FUNCTION "m7a_1_OF_4_BITS" : VOID
TITLE =1 AUS 4 Bits: lässt nur 1 von 4 Bits mit High-Signal zu
//1 AUS 4 Bits: lässt nur 1 von 4 Bits mit High-Signal zu. Das letzte Signal mit
//positiver Flanke bleibt jeweils erhalten, die anderen beiden werden
//zurückgesetzt.
//
//VERWENDUNG:
//Richtungs- bzw. Positions- Steuersignale aus Schrittketten. Somit muss nur der
//jeweils aktuelle Richtungsmerker gesetzt werden, ohne den alten Richtungsmerker
//zu löschen. Dies hilft Flüchtigkeitsfehler bei Programmierung zu vermeiden.
//
//z.B. hat man eine Bewegung die mit 2 ungleich langen Zylindern auf 4 Positionen
//gesteuert wird:
//Positionen LINKS, MITTE_LINKS, MITTE_RECHTS, RECHTS. Ohne Verwendung dieses FCs
//muß man bei einem
//Positionswchsel immer alle 3 Richtungsmerker bearbeiten
//  S LINKS
//  R MITTE_LINKS
//  R MITTE_RECHTS
//  R RECHTS
//Mit Verwendung dieses FCs entfällt das Rücksetzen, somit ergibt sich als
//Steuerprogramm für LINKS nur noch
//  S LINKS
//
//AUTOR: Stefan Maag, Dipl.-Ing. (FH) Elektrotechnik
//DATUM: 9/2004
//INTERNET: www.maagic7.de
//
//AENDERUNGSVERMERKE:
//--------------------------------------------------------------------------------
//DATUM        NAME        AENDERUNG
//--------------------------------------------------------------------------------
//21.04.2009   S.Maag      FC-ENO-Ausgang := ein Eingangsbit ist aktiv
//
//05.01.2015   S.Maag      Flankenmerker zusammen mit Bits löschen sonst können 2
//                         Bits aktiv werden, wenn ein gelöschtes Bit im gleichen
//                         CPU Zyklus sofort wieder gesetzt wird.
//                         (kommt normal nicht vor und wie man sieht ist es
//                         erst nach 10Jahren aufgefallen!)
//--------------------------------------------------------------------------------
//
//HINWEISE:
AUTHOR : 'S.Maag'
FAMILY : Maagic7
VERSION : 0.1


VAR_IN_OUT
  Bit1 : BOOL ;	//Merker 1
  Bit2 : BOOL ;	//Merker 2
  Bit3 : BOOL ;	//Merker 3
  Bit4 : BOOL ;	//Merker 4
  tmpByte : BYTE ;	//Hilfsbyte für Zustandsspeicherung
END_VAR
VAR_TEMP
  tmpBit1 : BOOL ;
  tmpBit2 : BOOL ;
  tmpBit3 : BOOL ;
  tmpBit4 : BOOL ;
  tmpBit5 : BOOL ;
  tmpBit6 : BOOL ;
  tmpBit7 : BOOL ;
  tmpBit8 : BOOL ;
END_VAR
BEGIN
NETWORK
TITLE =Hilfsbyte in lokalen Speicherbereich zur Bitadressierung

      L     #tmpByte;
      T     LB     0;
NETWORK
TITLE =Flanken der Bits prüfen und andere Bits löschen

      U     #Bit1; // Bit 1 auf positive Flanke prüfen
      FP    #tmpBit1;
      SPB   C234; // wenn ja, Bit 2/3/4 löschen

      U     #Bit2; // Bit 2 auf positive Flanke prüfen
      FP    #tmpBit2;
      SPB   C134; // wenn ja, Bit 1/3/4 löschen

      U     #Bit3;
      FP    #tmpBit3;
      SPB   C124;

      U     #Bit4;
      FP    #tmpBit4;
      SPB   C123;
      SPA   END;

C234: R     #Bit2; // CLR Bit 2/3/4
      R     #Bit3;
      R     #Bit4;
      R     #tmpBit2; // CLR Flankenmerker
      R     #tmpBit3; // CLR Flankenmerker
      R     #tmpBit4; // CLR Flankenmerker
      SPA   END;
C134: R     #Bit1; // CLR Bit 1/3/4
      R     #Bit3;
      R     #Bit4;
      R     #tmpBit1; // CLR Flankenmerker
      R     #tmpBit3; // CLR Flankenmerker
      R     #tmpBit4; // CLR Flankenmerker
      SPA   END;
C124: R     #Bit1; // CLR Bit 1/2/4
      R     #Bit2;
      R     #Bit4;
      R     #tmpBit1; // CLR Flankenmerker
      R     #tmpBit2; // CLR Flankenmerker
      R     #tmpBit4; // CLR Flankenmerker
      SPA   END;
C123: R     #Bit1; // CLR Bit 1/2/3
      R     #Bit2;
      R     #Bit3;
      R     #tmpBit1; // CLR Flankenmerker
      R     #tmpBit2; // CLR Flankenmerker
      R     #tmpBit3; // CLR Flankenmerker

NETWORK
TITLE =aktuelles Hilfsbyte wieder zurückschreiben

END:  L     LB     0;
      T     #tmpByte;

      O     #Bit1;
      O     #Bit2;
      O     #Bit3;
      O     #Bit4;
      SAVE  ;
      CLR   ;

END_FUNCTION

FUNCTION "m7a_CreateS5TimeFromINT" : VOID
TITLE =Minuten, Sekunden (im INT-Format) in das S5Time-Format wandeln
//Umwandlung von Minuten und/oder Sekunden in das S5Time-Format mit der
//gümstigsten Zeitbasis.
//Maximal sind mit dem S5Time-Format 9990sec möglich, das entspricht 2h46min30sec
//oder 166min 30sec
//
//AUTOR: Stefan Maag, Dipl.-Ing. (FH) Elektrotechnik
//DATUM: 9/2004
//INTERNET: www.maagic7.de
//
//AENDERUNGSVERMERKE:
//--------------------------------------------------------------------------------
//DATUM        NAME        AENDERUNG
//--------------------------------------------------------------------------------
//24.01.2005   S.Maag    Fehler BCD Wandlung bei Zeitbasis 10sec behoben
//--------------------------------------------------------------------------------
//
//HINWEISE:
AUTHOR : 'S.Maag'
FAMILY : Maagic7
VERSION : 0.1


VAR_INPUT
  MIN : INT ;	//Anzahl Minuten (max = 166min, da S5MaxTime=9990sec)
  SEC : INT ;	//Anzahl Sekunden
END_VAR
VAR_OUTPUT
  S5_TIME : S5TIME ;
END_VAR
BEGIN
NETWORK
TITLE =Umwandlung in die günstigste Zeitbasis
//S5Time-Format Bits:
//
//15 | 14 | 13 | 12 | 11 | 10 | 9 | 8 | 7 | 6 | 5 | 4 | 3 | 2 | 1 | 0
//  x   x | Zeitbas.|             Zeitwert im BCD Format
//
//Zeitbasis : Bits fuer Zeitbasis
//     10ms : 00
//    100ms : 01
//      1s  : 10
//     10s  : 11
      L     #MIN; // Minuten
      L     60; // Sekunden/Minute
      *I    ; // Sekunden von Minuten
      L     #SEC; // Sekunden
      +I    ; // Sekunden gesamt
      L     9; // bis 9 Sekunden
      TAK   ; // Sekunden in Akku 1, Vergleichswert in Akku 2
      >=I   ;
      SPB   hdst; // Zeitbasis 10ms = 1/100sec

      L     99; // bis 99 Sekunden
      TAK   ;
      >=I   ;
      SPB   zntl; // Zeitbasis 100ms = 1/10sec

      L     990; // bis 990 Sekunden
      TAK   ;
      >=I   ;
      SPB   sec; // Zeitbasis 1 Sekunde

      L     9990;
      TAK   ;
      >=I   ; // falls nicht mehr als 9990 Sekunden, dann
      SPB   zehn; // Zeitbasis Zehn Sekunden
      TAK   ; // sonst Begrenzung: 9990 wieder in Akku 1

zehn: L     10; // zuerst durch 10 teilen, da  Werte > 999 nicht mit
      /I    ; // dem ITB Befehl in BCD gewandelt werden können. Ein SRW 4 der
      ITB   ; // BCD Zahl geht hier nicht, da die Sekunden > 999 sein können.
      L     W#16#3000; // Zeitbasis Zehn Sekunden
      OW    ; // Bits für Zeitbasis einblenden
      SPA   SAVE;

sec:  ITB   ; // Anzahl der Sekunden ins BCD Format
      L     W#16#2000; // Zeitbasis Sekunden
      OW    ; // Bits für Zeitbasis einblenden
      SPA   SAVE;

zntl: ITB   ; // Anzahl der Sekunden (max, 999) ins BCD Format
      SLW   4; // 4 Bits nach links := 1 Stelle im 10er BCD Format := *10
      L     W#16#1000; // Zeitbasis 10ms
      OW    ; // Bits für Zeitbasis einblenden
      SPA   SAVE;

hdst: ITB   ; // Anzahl der Sekunden ins BCD Format
      SLW   8; // 8 Bits nach links := 2 Stellen im 10er BCD Format := *100
      L     W#16#0; // Zeitbasis 100ms
      OW    ; // Bits für Zeitbasis einblenden
SAVE: T     #S5_TIME; // Zeit im S5Time-Format
NETWORK
TITLE =FC-ENO

      SET   ;
      SAVE  ;
      CLR   ;

END_FUNCTION

FUNCTION "m7a_CreateIECTimeFromINT" : VOID
TITLE =Time hh:mm:ss [INT] to IEC TIME
//AUTOR: Stefan Maag, Dipl.-Ing. (FH) Elektrotechnik
//DATUM: 9/2004
//INTERNET: www.maagic7.de
//
//AENDERUNGSVERMERKE:
//--------------------------------------------------------------------------------
//DATUM        NAME        AENDERUNG
//--------------------------------------------------------------------------------
//20.03.2018   S.Maag      changed from mm:ss to hh:mm:ss
//--------------------------------------------------------------------------------
//
//HINWEISE:
AUTHOR : 'S.Maag'
FAMILY : Maagic7
VERSION : 0.1


VAR_INPUT
  hh : INT ;	//Hours
  mm : INT ;	//Minutes
  ss : INT ;	//Seconds
END_VAR
VAR_OUTPUT
  IEC_TIME : TIME ;
END_VAR
VAR_TEMP
  dMilliSeconds : DINT ;	//Sekunden als Millisekunden
END_VAR
BEGIN
NETWORK
TITLE =ss to milli seconds

      L     #ss; // seconds
      ITD   ; // to DINT
      L     L#1000; // 1sec = 1000ms
      *D    ;
      T     #dMilliSeconds; // save

NETWORK
TITLE =Minutes to milli seconds

      L     #mm; // Minutes
      ITD   ; // to DINT
      L     L#60000; // 1 min = 60000ms
      *D    ;
      L     #dMilliSeconds;
      +D    ;
      T     #dMilliSeconds;

NETWORK
TITLE =hours to milli seconds

      L     #hh; // hours
      ITD   ; // to DINT
      L     L#3600000; // 1h = 3600.000ms
      *D    ;
      L     #dMilliSeconds;
      +D    ;
      T     #IEC_TIME;

NETWORK
TITLE =FC-ENO-Ausgang

      SET   ;
      SAVE  ;
      CLR   ;

END_FUNCTION

FUNCTION "m7a_INV_IEC_TIME" : VOID
TITLE =IEC Zeit invertieren, Rückwärtszählung
//IEC Zeit invertieren. Wird benötigt z.B. benötigt, wenn Ausschaltverzögerungen
//über SFB5 programmiert werden und die Zeitanzeige dann rückwärts laufen soll.
//SFB5 stellt nur einen vorwärts laufenden Timerwert zur Verfügung
//
//AUTOR: Stefan Maag, Dipl.-Ing. (FH) Elektrotechnik
//DATUM: 1/2005
//INTERNET: www.maagic7.de
//
//AENDERUNGSVERMERKE:
//--------------------------------------------------------------------------------
//DATUM        NAME            AENDERUNG
//--------------------------------------------------------------------------------
//
//--------------------------------------------------------------------------------
//
//HINWEISE:
AUTHOR : 'S.Maag'
FAMILY : Maagic7
VERSION : 0.1


VAR_INPUT
  iecDauer : TIME ;	//Dauer
  iecTimer : TIME ;	//Zeitwert vom Timer
END_VAR
VAR_OUTPUT
  iecInvTime : TIME ;
END_VAR
BEGIN
NETWORK
TITLE =

      L     #iecDauer;
      L     #iecTimer;
      -D    ;
      L     L#0;
      <D    ;
      SPB   SAVE;
      TAK   ;
SAVE: T     #iecInvTime;
NETWORK
TITLE =FC-ENO

      SET   ;
      SAVE  ;
      CLR   ;

END_FUNCTION

FUNCTION "m7a_DINT_MM.SS_TO_IEC" : VOID
TITLE =Zeit DINT MM.SS in das IEC-Zeitformat wandeln
//AUTOR: Stefan Maag, Dipl.-Ing. (FH) Elektrotechnik
//DATUM: 1/2005
//INTERNET: www.maagic7.de
//
//AENDERUNGSVERMERKE:
//--------------------------------------------------------------------------------
//DATUM        NAME       AENDERUNG
//--------------------------------------------------------------------------------
//22.04.2014   S.Maag     Ausgang IEC-Zeit auf min. 1ms begrenzt, da 0ms = RESET
//--------------------------------------------------------------------------------
//
//HINWEISE:
AUTHOR : 'S.Maag'
FAMILY : Maagic7
VERSION : 0.1


VAR_OUTPUT
  IEC_TIME : TIME ;
END_VAR
VAR_IN_OUT
  MM_SS : DINT ;	//Minuten und Sekunden z.B.: 0530 = 5m30s
END_VAR
VAR_TEMP
  MM : DINT ;	//Minutenwert
  SS : DINT ;	//Sekundenwert
  SS_msec : DINT ;	//Sekunden als Millisekunden
END_VAR
BEGIN
NETWORK
TITLE =Minuten und Sekundenanteil aus MM.SS lösen

      L     #MM_SS; // Minuten.Sekunden
      L     L#100;
      MOD   ; // Modulo Division
      T     #SS; // =Divisionsrest = Sekunden

      L     #MM_SS;
      L     L#100;
      /D    ;
      T     #MM;

NETWORK
TITLE =Sekundenanteil in Millisekunden umrechnen

      L     #SS; // Sekunden
      L     1000;
      *D    ;
      T     #SS_msec; // Millisekunden

NETWORK
TITLE =Minutenanteil in Millisekunden umrechnen
//22.04.2014 IEC-Zeit auf min. 1ms begrenzt, da 0ms = RESET
      L     #MM; // Minuten
      L     L#60000; // Millisekunden pro Minute
      *D    ;
      L     #SS_msec; // Anteil der Sekunden
      +D    ; // + Anteil der Minuten
      U     >0;
      SPB   save;
      L     L#1;
save: T     #IEC_TIME; // ergibt gesamte Millisekunden

NETWORK
TITLE =Wenn Sekunden >59, dann 1 Minute dazu und Sekunden anpassen

      L     #SS; // Sekundenwert
      L     59; // prüfen, ob weniger als 60
      <=D   ; // Sekunden, dann o.k.
      SPB   NE4;

      L     #MM_SS; // Minuten.Sekunden laden
      +     L#40; // Wenn mehr als 60Sekunden, dann müssen die fehlenden
      T     #MM_SS; // 40 Sekunden für den Überlauf dazugezählt werden
NE4:  NOP   0;

NETWORK
TITLE =FC-ENO-Ausgang

      SET   ;
      SAVE  ;
      CLR   ;

END_FUNCTION

FUNCTION "m7a_IEC_TO_MM.SS_DINT" : VOID
TITLE =IEC Zeit in DINT MM.SS wandeln
//AUTOR: Stefan Maag, Dipl.-Ing. (FH) Elektrotechnik
//DATUM: 1/2005
//INTERNET: www.maagic7.de
//
//AENDERUNGSVERMERKE:
//--------------------------------------------------------------------------------
//DATUM        NAME            AENDERUNG
//--------------------------------------------------------------------------------
//
//--------------------------------------------------------------------------------
//
//HINWEISE:
AUTHOR : 'S.Maag'
FAMILY : Maagic7
VERSION : 0.1


VAR_INPUT
  IEC_TIME : TIME ;
END_VAR
VAR_OUTPUT
  MM_SS : DINT ;
END_VAR
VAR_TEMP
  MM : DINT ;	//Minutenwert
  SS : DINT ;	//Sekundenwert
END_VAR
BEGIN
NETWORK
TITLE =Minuten- und Sekundenanteil

      L     #IEC_TIME;
      L     L#60000; // Millisekunden pro Minute
      /D    ;
      T     #MM; // Minuten

      L     #IEC_TIME;
      L     L#60000; // Millisekunden pro Minute
      MOD   ; // Restwerdivision: Rest ms
      L     L#1000;
      /D    ; // Modulo Division
      T     #SS; // =Divisionsrest = Sekunden

      L     #MM; // Minuten*100
      L     L#100;
      *D    ;
      L     #SS;
      +D    ;
      T     #MM_SS; // Wert in MM.SS

NETWORK
TITLE =FC-ENO-Ausgang

      SET   ;
      SAVE  ;
      CLR   ;

END_FUNCTION

FUNCTION "m7a_DINT_MM.SS_TO_S5Time" : VOID
TITLE =Zeit DINT MM.SS in das S5-Zeitformat wandeln
//Zeiten werden als DINT-Wert mit 2 Nachkommastellen eingegeben, welche den
//Sekunden entsprechen. Die Minuten sind der Wert vor dem Komma. Werden Sekunden
//größer als 59 eingegebn, so werden diese automatisch auf Minuten umgerechnet
//und der eingegebene Wert MM.SS richtig angepasst.
//
//AUTOR: Stefan Maag, Dipl.-Ing. (FH) Elektrotechnik
//DATUM: 1/2005
//INTERNET: www.maagic7.de
//
//AENDERUNGSVERMERKE:
//--------------------------------------------------------------------------------
//DATUM        NAME            AENDERUNG
//--------------------------------------------------------------------------------
//
//--------------------------------------------------------------------------------
//
//HINWEISE:
AUTHOR : 'S.Maag'
FAMILY : Maagic7
VERSION : 0.1


VAR_OUTPUT
  S5_Time : S5TIME ;
END_VAR
VAR_IN_OUT
  MM_SS : DINT ;	//Minuten und Sekunden z.B.: 0530 = 5m30s
END_VAR
VAR_TEMP
  MM : INT ;	//Minutenwert
  SS : INT ;	//Sekundenwert
END_VAR
BEGIN
NETWORK
TITLE =Minuten und Sekundenanteil aus MM.SS lösen

      L     #MM_SS; // Minuten.Sekunden
      L     L#100;
      MOD   ; // Modulo Division
      T     #SS; // =Divisionsrest = Sekunden

      L     #MM_SS;
      L     L#100;
      /D    ;
      T     #MM;

NETWORK
TITLE =Wenn Sekunden >59, dann 1 Minute dazu und Sekunden anpassen

      L     #SS; // Sekundenwert
      L     59; // prüfen, ob weniger als 60
      <=D   ; // Sekunden, dann o.k.
      SPB   NE4;

      L     #MM_SS; // Minuten.Sekunden laden
      +     L#40; // Wenn mehr als 60Sekunden, dann müssen die fehlenden
      T     #MM_SS; // 40 Sekunden für den Überlauf dazugezählt werden
NE4:  NOP   0;

NETWORK
TITLE =Umwandlung in die günstigste Zeitbasis
//S5Time-Format Bits:
//
//15 | 14 | 13 | 12 | 11 | 10 | 9 | 8 | 7 | 6 | 5 | 4 | 3 | 2 | 1 | 0
//  x   x | Zeitbas.|             Zeitwert im BCD Format
//
//Zeitbasis : Bits fuer Zeitbasis
//     10ms : 00
//    100ms : 01
//      1s  : 10
//     10s  : 11
      L     #MM; // Minuten
      L     60; // Sekunden/Minute
      *D    ; // Sekunden von Minuten
      L     #SS; // Sekunden
      +D    ; // Sekunden gesamt
      L     9; // bis 9 Sekunden
      TAK   ; // Sekunden in Akku 1, Vergleichswert in Akku 2
      >=I   ;
      SPB   hdst; // Zeitbasis 10ms = 1/100sec

      L     99; // bis 99 Sekunden
      TAK   ;
      >=I   ;
      SPB   zntl; // Zeitbasis 100ms = 1/10sec

      L     990; // bis 990 Sekunden
      TAK   ;
      >=I   ;
      SPB   sec; // Zeitbasis 1 Sekunde

      L     9990;
      TAK   ;
      >=I   ; // falls nicht mehr als 9990 Sekunden, dann
      SPB   zehn; // Zeitbasis Zehn Sekunden
      TAK   ; // sonst Begrenzung: 9990 wieder in Akku 1

zehn: L     10; // zuerst durch 10 teilen, da  Werte > 999 nicht mit
      /I    ; // dem ITB Befehl in BCD gewandelt werden können. Ein SRW 4 der
      ITB   ; // BCD Zahl geht hier nicht, da die Sekunden > 999 sein können.
      L     W#16#3000; // Zeitbasis Zehn Sekunden
      OW    ; // Bits für Zeitbasis einblenden
      SPA   SAVE;

sec:  ITB   ; // Anzahl der Sekunden ins BCD Format
      L     W#16#2000; // Zeitbasis Sekunden
      OW    ; // Bits für Zeitbasis einblenden
      SPA   SAVE;

zntl: ITB   ; // Anzahl der Sekunden (max, 999) ins BCD Format
      SLW   4; // 4 Bits nach links := 1 Stelle im 10er BCD Format := *10
      L     W#16#1000; // Zeitbasis 10ms
      OW    ; // Bits für Zeitbasis einblenden
      SPA   SAVE;

hdst: ITB   ; // Anzahl der Sekunden ins BCD Format
      SLW   8; // 8 Bits nach links := 2 Stellen im 10er BCD Format := *100
      L     W#16#0; // Zeitbasis 100ms
      OW    ; // Bits für Zeitbasis einblenden
SAVE: T     #S5_Time; // Zeit im S5Time-Format
NETWORK
TITLE =FC-ENO-Ausgang

      SET   ;
      SAVE  ;
      CLR   ;

END_FUNCTION

FUNCTION "m7a_MMSS_BCD_TO_IEC" : VOID
TITLE =Zeit hexadezimal MM.SS in das IEC-Zeitformat wandeln
//AUTOR: Stefan Maag, Dipl.-Ing. (FH) Elektrotechnik
//DATUM: 10/2004
//INTERNET: www.maagic7.de
//
//AENDERUNGSVERMERKE:
//--------------------------------------------------------------------------------
//DATUM        NAME        AENDERUNG
//--------------------------------------------------------------------------------
//
//--------------------------------------------------------------------------------
//
//HINWEISE:
AUTHOR : 'S.Maag'
FAMILY : Maagic7
VERSION : 0.1


VAR_INPUT
  MIN_BCD : BYTE ;	//Minuten als BCD-Wert
  SEC_BCD : BYTE ;	//Sekunden als BCD-Wert
END_VAR
VAR_OUTPUT
  IEC_TIME : TIME ;
END_VAR
VAR_TEMP
  SS_msec : DINT ;	//Sekunden als Millisekunden
END_VAR
BEGIN
NETWORK
TITLE =Sekundenanteil in Millisekunden umrechen

      L     #SEC_BCD; // Sekunden im HEX-Format
      SLD   12; // * 1000 = Millisekunden
      BTD   ; // BCD->DINT
      T     #SS_msec; // zwischenspeichern

NETWORK
TITLE =Minutenanteil in Millisekunden umrechnen

      L     #MIN_BCD; // Minuten im HEX-Format
      SLD   12; // *1000
      BTD   ; // BCD->DINT
      L     L#60; // Sekunden pro Minute
      *D    ; // *1000 *60 := Millisekunden
      L     #SS_msec; // Anteil der Sekunden
      +D    ; // + Anteil der Minuten
      T     #IEC_TIME; // ergibt gesamte Millisekunden

NETWORK
TITLE =FC-ENO-Ausgang

      SET   ;
      SAVE  ;
      CLR   ;

END_FUNCTION

FUNCTION "m7a_ZeitDauer" : VOID
TITLE =Zeitdauer Abgelaufen?
//Überprüft, ob seit der übergebenen Startzeit die gewünschte Dauer abgelaufen
//ist. Die Zeiten werden im IEC-TIME-FORMAT übergeben
//
//BENÖTIGTE SFCs: SFC1 - READ_CLK
//
//AUTOR: Stefan Maag, Dipl.-Ing. (FH) Elektrotechnik
//DATUM: 9/2004
//INTERNET: www.maagic7.de
//
//AENDERUNGSVERMERKE:
//--------------------------------------------------------------------------------
//DATUM        NAME        AENDERUNG
//--------------------------------------------------------------------------------
//03/12/2013   S.Maag      SFC64 TimeTick Zeitdifferenz korrigiert
//                         da 31Bit, Fehler bei Überlauf. Jetzt UC FC256
//--------------------------------------------------------------------------------
//
//HINWEISE:
AUTHOR : 'S.Maag'
FAMILY : Maagic7
VERSION : 0.1


VAR_INPUT
  START_ZEIT : TIME ;
  DAUER : TIME ;
END_VAR
VAR_OUTPUT
  OUT_TIMER : BOOL ;	//TimerAusgang: Zeit abgelaufen
  TIME_LEFT : TIME ;	//Restlaufzeit
END_VAR
VAR_TEMP
  aktSysTime : TIME ;	//aktuelle Systemzeit
END_VAR
BEGIN
NETWORK
TITLE =aktuelle SystemZeit auslesen

      CALL "TIME_TCK" (
           RET_VAL                  := #aktSysTime);
      NOP   0;

NETWORK
TITLE =prüfen ob Zeit abgelaufen ist

      L     #START_ZEIT;
      L     #aktSysTime;
      UC    "m7b_ABS_DIFF_S7SysTime"; // Absolute Differenz S7SytemTimer 31Bit
      L     #DAUER;
      >D    ;
      =     #OUT_TIMER;
      SAVE  ;
      TAK   ;
      -D    ;
      T     #TIME_LEFT;

END_FUNCTION

FUNCTION "m7a_CreateANY" : VOID
TITLE =CreateANY: erzeugt ANY aus Einzelbestandteilen
//Codierung Datentyp:
//00h : NIL  : Nullpointer
//01h : BOOL : Bits
//02h : BYTE
//03h : CHAR
//04h : WORD
//05h : INT
//06h : DWORD
//07h : DINT
//08h : REAL
//09h : DATE
//0Ah : Time_OF_DAY (TOD)
//0Bh : TIME
//0Ch : S5Time
//0Dh : nicht definiert
//0Eh : DATE_AND_TIME (DT)
//13h : STRING
//
//Codierung Speicherbereich:
//80h : P : Peripherie
//81h : E : Eingänge
//82h : A : Ausgänge
//83h : M : Merker
//84h : DB: Datenbaustein
//85h : DI: Instanzdatenbaustein
//86h : L : Lokaldaten (L-Stack)
//87h : V : voriger Lokaldatenstack
//
//AUTOR: Stefan Maag, Dipl.-Ing. (FH) Elektrotechnik
//DATUM: 10/2007
//INTERNET: www.maagic7.de
//
//AENDERUNGSVERMERKE:
//--------------------------------------------------------------------------------
//DATUM        NAME       AENDERUNG
//--------------------------------------------------------------------------------
//04.11.2011   S.Maag     Fehler Speicherbereichsverarbeitung mit UD statt OD
//                        behoben
//--------------------------------------------------------------------------------
//
//HINWEISE:
AUTHOR : 'S.Maag'
FAMILY : Maagic7
VERSION : 0.1


VAR_INPUT
  B1_DataType : BYTE ;	//1=Bool 2=Byte 3=Char 4=Word 5=INT 6=DW 7=DINT 8=Real 9=Date ...
  B23_Wiederholung : INT ;	//Wiederholungsfaktor
  B45_DB : INT ;	//DB-Nummer oder 0
  B6_Speicher : BYTE ;	//Hex 80=P 81=E 82=A 83=M 84=DB 85=DI 86=L 87=V
  ByteAdr : INT ;	//ByteAdresse
  BitAdr : INT ;	//Bitadresse 0..7
END_VAR
VAR_OUTPUT
  AnyPointer : ANY ;
END_VAR
VAR_TEMP
  pBit : DWORD ;
  AR1 : DWORD ;
END_VAR
BEGIN
NETWORK
TITLE =

      L     P##AnyPointer;
      LAR1  ;
// Byte 0 enthält immer 10h für S7
      L     B#16#10;
      T     B [AR1,P#0.0];

      L     #B1_DataType;
      T     B [AR1,P#1.0]; // Byte 1 = Datentyp

      L     #B23_Wiederholung;
      T     W [AR1,P#2.0]; // Byte 2&3 = Wiederholungsfaktor

      L     #B45_DB;
      T     W [AR1,P#4.0]; // Byte 4&5 = Datenbaustein-Nr

      L     #BitAdr;
      L     B#16#7; // Bitadresse auf 3 Bit Begrenzen 0..7
      UW    ;
      L     #ByteAdr; // ByteAdresse um 3 nach links => Pointerformat
      SLD   3;
      OD    ; // ByteAdress und Bitadresse verbinden
      T     D [AR1,P#6.0];

      L     #B6_Speicher;
      T     B [AR1,P#6.0]; // Byte 6 = Speicherbereich

      SET   ;
      SAVE  ;
      CLR   ;
END_FUNCTION

FUNCTION "m7a_SplitAny" : VOID
TITLE =SplitAny : Zerteilt ANY-Pointer in die relevanten Bestandteile
//Codierung Datentyp:
//00h : NIL  : Nullpointer
//01h : BOOL : Bits
//02h : BYTE
//03h : CHAR
//04h : WORD
//05h : INT
//06h : DWORD
//07h : DINT
//08h : REAL
//09h : DATE
//0Ah : Time_OF_DAY (TOD)
//0Bh : TIME
//0Ch : S5Time
//0Dh : nicht definiert
//0Eh : DATE_AND_TIME (DT)
//13h : STRING
//
//Codierung Speicherbereich:
//80h : P : Peripherie
//81h : E : Eingänge
//82h : A : Ausgänge
//83h : M : Merker
//84h : DB: Datenbaustein
//85h : DI: Instanzdatenbaustein
//86h : L : Lokaldaten (L-Stack)
//87h : V : voriger Lokaldatenstack
//
//AUTOR: Stefan Maag, Dipl.-Ing. (FH) Elektrotechnik
//DATUM: 10/2007
//INTERNET: www.maagic7.de
//
//AENDERUNGSVERMERKE:
//--------------------------------------------------------------------------------
//DATUM        NAME            AENDERUNG
//--------------------------------------------------------------------------------
//
//--------------------------------------------------------------------------------
//
//HINWEISE:
AUTHOR : 'S.Maag'
FAMILY : Maagic7
VERSION : 0.1


VAR_INPUT
  AnyPointer : ANY ;
END_VAR
VAR_OUTPUT
  B1_DataType : BYTE ;
  B23_Wiederholung : INT ;
  B45_DB : INT ;
  B6_Speicher : BYTE ;
  ByteAdr : INT ;
  BitAdr : INT ;
END_VAR
VAR_TEMP
  AR1 : DWORD ;
END_VAR
BEGIN
NETWORK
TITLE =

      TAR1  #AR1; // Adressregister 1 sichern

      L     P##AnyPointer;
      LAR1  ;
// Byte 0 enthält immer 10h für S7, daher nicht ausgeben
// L     B [AR1,P#0.0]
// T     #B0_PLC

      L     B [AR1,P#1.0]; // Byte 1 = Datentyp
      T     #B1_DataType;

      L     W [AR1,P#2.0]; // Byte 2&3 = Wiederholungsfaktor
      T     #B23_Wiederholung;

      L     W [AR1,P#4.0]; // Byte 4&5 = Datenbaustein-Nr
      T     #B45_DB;

      L     B [AR1,P#6.0]; // Byte 6 = Speicherbereich
      T     #B6_Speicher;

      L     D [AR1,P#6.0]; // Byte 7&8&9 = BitPointer
      SRD   3; // daraus ByteAdresse berechnen
      T     #ByteAdr;

      L     B [AR1,P#9.0]; // Byte 9, Bit 0..2 = Bitadresse
      L     B#16#7;
      UW    ;
      T     #BitAdr;

      LAR1  #AR1; // ursprüngliches Adressregister 1 herstellen
      SET   ;
      SAVE  ;
      CLR   ;
END_FUNCTION

FUNCTION "m7a_SternDreieck" : VOID
TITLE =Stern- Dreieck- Anlauf
//Stern-Dreieck Anlauf
//
//IN:
//START: Stern-Dreieck Anlauf Einschalten
//FRG  : Freigabe
//T_STERN: Stern Anlaufzeit im S5 Zeitformat
//TIMER_S5: Timer im S5-Format
//
//InOut:
//bTmp:  externes dauerhaftes Speicherbyte für Hilfsignale
//
//OUT:
//NETZ:    Netz-Schütz
//DREIECK: Dreick-Schütz
//STERN:   Stern-Schütz
//
//AUTOR: Stefan Maag, Dipl.-Ing. (FH) Elektrotechnik
//DATUM: 01/2006
//INTERNET: www.maagic7.de
//
//AENDERUNGSVERMERKE:
//--------------------------------------------------------------------------------
//DATUM        NAME            AENDERUNG
//--------------------------------------------------------------------------------
//
//--------------------------------------------------------------------------------
//
//HINWEISE:
AUTHOR : 'S.Maag'
FAMILY : Maagic7
VERSION : 0.1


VAR_INPUT
  START : BOOL ;
  FRG : BOOL ;	//Freigabe
  T_STERN : S5TIME ;
  TIMER_S5 : TIMER ;
END_VAR
VAR_OUTPUT
  NETZ : BOOL ;	//Netzschütz
  DREIECK : BOOL ;	//Dreieckschütz
  STERN : BOOL ;	//Sternbrücke
END_VAR
VAR_IN_OUT
  bTmp : BYTE ;
END_VAR
VAR_TEMP
  lb_NETZ : BOOL ;
  lb_DREIECK : BOOL ;
  lb_STERN : BOOL ;
  lb3 : BOOL ;
  lb4 : BOOL ;
  lb5 : BOOL ;
  lb6 : BOOL ;
  lb7 : BOOL ;
END_VAR
BEGIN
NETWORK
TITLE =



NETWORK
TITLE =Speichervariable in Lokaldaten
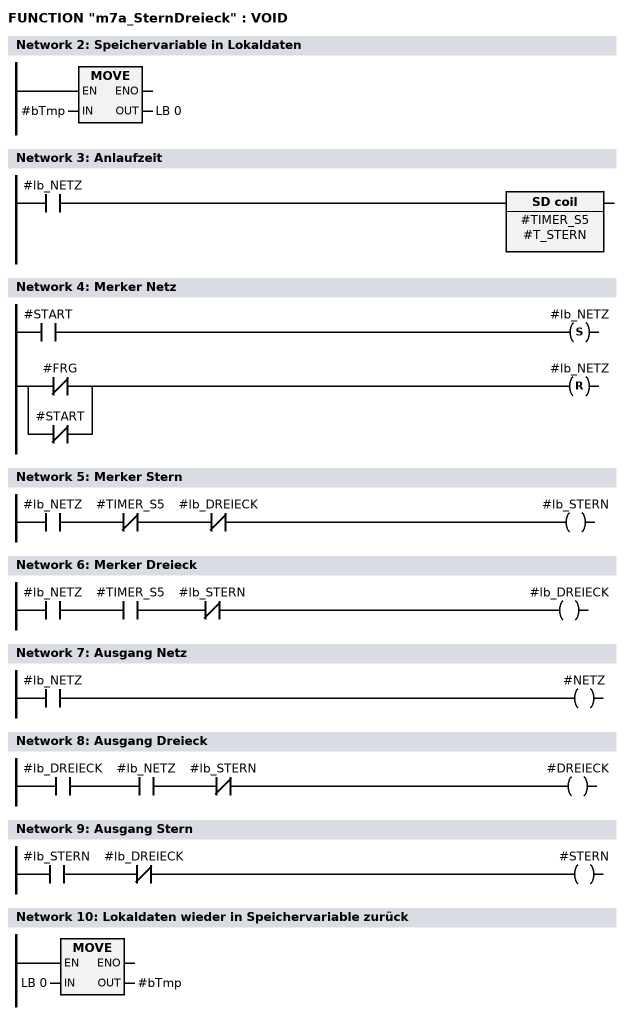

      L     #bTmp;
      T     LB     0;


NETWORK
TITLE =Anlaufzeit



      U     #lb_NETZ;
      L     #T_STERN;
      SE    #TIMER_S5;
      NOP   0;
      NOP   0;
      NOP   0;
      NOP   0;
NETWORK
TITLE =Merker Netz

      U     #START;
      S     #lb_NETZ;
      U(    ;
      ON    #FRG;
      ON    #START;
      )     ;
      R     #lb_NETZ;
      NOP   0;
NETWORK
TITLE =Merker Stern

      U     #lb_NETZ;
      UN    #TIMER_S5;
      UN    #lb_DREIECK;
      =     #lb_STERN;
NETWORK
TITLE =Merker Dreieck

      U     #lb_NETZ;
      U     #TIMER_S5;
      UN    #lb_STERN;
      =     #lb_DREIECK;
NETWORK
TITLE =Ausgang Netz

      U     #lb_NETZ;
      =     #NETZ;
NETWORK
TITLE =Ausgang Dreieck

      U     #lb_DREIECK;
      U     #lb_NETZ;
      UN    #lb_STERN;
      =     #DREIECK;
NETWORK
TITLE =Ausgang Stern

      U     #lb_STERN;
      UN    #lb_DREIECK;
      =     #STERN;
NETWORK
TITLE =Lokaldaten wieder in Speichervariable zurück

      L     LB     0;
      T     #bTmp;

END_FUNCTION

FUNCTION "m7a_WendeSchuetz" : VOID
TITLE =Sichere Wendeschützschaltung mit Speicherung des Schaltzustands
//Sichere Wendeschützschaltung mit Umschaltverzögerung:
//
//Über den Eingang Save kann angegeben werden, dass der aktuelle Schaltzustand
//bis zum nächsten Richtungswechsel gespeichert/geschaltet bleibt. Werden beide
//Richtungseingänge geschaltet, werden die Ausgänge sofort gelöscht. Sind beide
//Richtung aktiv, z.B. durch setzen des Richtungsmerkers ausserhalb des FCs, so
//wird die Linksdrehrichtung abgeschaltet.
//
//Der FC-ENO Ausgang ist "1", solange ein Richtungsausgang aktiv ist.
//
//SAVE = 1 :  Der Richtungsausgang bleibt solange geschaltet, bis der andere
//            Richtungsbefehl anliegt. Es wird dann mit der Verzögerung T
//            umgeschaltet. Diesen Modus kann man nur verwenden, wenn ein
//            vorgeschaltetes Gerät wie z.B. Spannungssteller den Motor
//            abschaltet.
//
//SAVE = 0 :  Der Richtungsausgang bleibt immer nur solange erhalten wie der
//            entsprechende Richtungseingang anliegt. Das Umschalten der
//            Richtungsausgänge wird dabei mit T verzögert.
//
//AUTOR: Stefan Maag, Dipl.-Ing. (FH) Elektrotechnik
//DATUM: 3/2003
//INTERNET: www.maagic7.de
//
//AENDERUNGSVERMERKE:
//--------------------------------------------------------------------------------
//DATUM        NAME            AENDERUNG
//--------------------------------------------------------------------------------
//
//--------------------------------------------------------------------------------
//12/2004    S.Maag     Richtungssignal vorhanden, auf FC-ENO Ausgang verschaltet.
//
//                      Verriegelung, so daß nur 1 Richtungssignal aktiv sein kann
//
//
//HINWEISE:
AUTHOR : 'S.Maag'
FAMILY : Maagic7
VERSION : 0.1


VAR_INPUT
  RECHTS : BOOL ;	//Richtung vorwärts
  LINKS : BOOL ;	//Richtung rückwärts
  SAVE : BOOL ;	//=0 : (Ausgang=Eingangssignal); =1:(Ausgang wird gesetzt)
  T : TIMER ;	//Zeitglied
  T_S5 : S5TIME ;	//Zeitwert Umschaltverzögerung
END_VAR
VAR_IN_OUT
  OUT_R : BOOL ;
  OUT_L : BOOL ;
END_VAR
BEGIN
NETWORK
TITLE =Ausgang für Richtung vorwärts/rechts
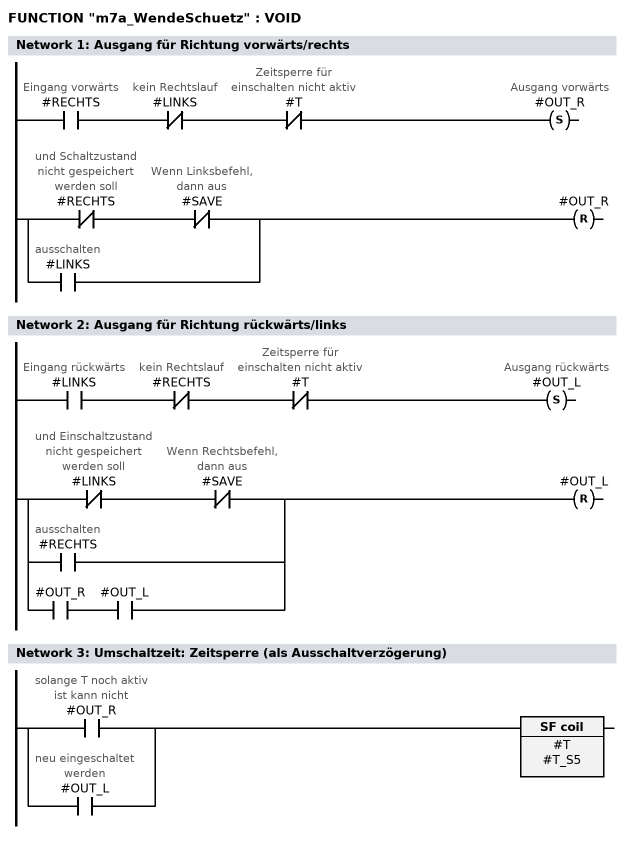


      U     #RECHTS; // Eingang vorwärts
      UN    #LINKS; // kein Rechtslauf
      UN    #T; // Zeitsperre für einschalten nicht aktiv
      S     #OUT_R; // Ausgang vorwärts
      U(    ; // Ausschalten wenn Richtung rechts nicht vorhanden
      UN    #RECHTS; // und Schaltzustand nicht gespeichert werden soll
      UN    #SAVE; // Wenn Linksbefehl, dann aus
      O     #LINKS; // ausschalten
      )     ;
      R     #OUT_R;
      NOP   0;
NETWORK
TITLE =Ausgang für Richtung rückwärts/links

      U     #LINKS; // Eingang rückwärts
      UN    #RECHTS; // kein Rechtslauf
      UN    #T; // Zeitsperre für einschalten nicht aktiv
      S     #OUT_L; // Ausgang rückwärts
      U(    ; // Ausschalten wenn Richtung rechts nicht vorhanden
      UN    #LINKS; // und Einschaltzustand nicht gespeichert werden soll
      UN    #SAVE; // Wenn Rechtsbefehl, dann aus
      O     #RECHTS; // ausschalten
      O     ;
      U     #OUT_R;
      U     #OUT_L;
      )     ;
      R     #OUT_L;
      NOP   0;
NETWORK
TITLE =Umschaltzeit: Zeitsperre (als Ausschaltverzögerung)

      U(    ; // Nachlauf der Richtungsausgänge,
      O     #OUT_R; // solange T noch aktiv ist kann nicht
      O     #OUT_L; // neu eingeschaltet werden
      )     ;
      L     #T_S5;
      SA    #T;
      NOP   0;
      NOP   0;
      NOP   0;
      NOP   0;
NETWORK
TITLE =FC-ENO Ausgang

      O     #OUT_R;
      O     #OUT_L;
      SAVE  ;
      CLR   ;
END_FUNCTION

FUNCTION "m7a_CompareANY" : VOID
TITLE =Compares 2 ANY-Pointer
//[IN]
//ANY1 : ANY-Pointer 1
//ANY2 : ANY-Pointer 2
//
//[RET]
//ENO  : TRUE if equal
//
//AUTOR: Stefan Maag, Dipl.-Ing. (FH) Elektrotechnik
//DATUM: 10/2010
//INTERNET: www.maagic7.de
//
//AENDERUNGSVERMERKE:
//--------------------------------------------------------------------------------
//DATUM        NAME            AENDERUNG
//--------------------------------------------------------------------------------
//
//--------------------------------------------------------------------------------
AUTHOR : 'S.Maag'
FAMILY : Maagic7
VERSION : 0.1


VAR_INPUT
  ANY1 : ANY ;
  ANY2 : ANY ;
END_VAR
VAR_TEMP
  AR1 : DWORD ;
END_VAR
BEGIN
NETWORK
TITLE =Adressregiste 1 sichern
//Adressregister 2 Global- und Instanz DB werden bei CALL-Aufrufen automatisch
//vom System gesichert, bei UC nicht!
      TAR1  #AR1; // Adressregister 1 sichern

NETWORK
TITLE =ANY-Pointer vergleichen
//Ein ANY umfasst 10Bytes
      L     P##ANY1; // Pointer to INPUT Variable ANY1
      LAR1  ;

      L     P##ANY2; // Pointer fo INPUT Variable ANY2
      LAR2  ;

      L     D [AR1,P#0.0]; // Byte 0..3
      L     D [AR2,P#0.0];
      <>D   ;
      SPB   NEQ; // not equal
      L     D [AR1,P#4.0]; // Byte 4..7
      L     D [AR2,P#4.0];
      <>D   ;
      SPB   NEQ; // not equal
      L     W [AR1,P#8.0]; // Byte 8..9
      L     W [AR2,P#8.0];
      <>D   ;
      SPB   NEQ; // not equal

      SAVE  ; // Wenn gleich
      SPA   END;

NEQ:  CLR   ; // Daten sind ungleich
      SAVE  ;

NETWORK
TITLE =Adressregister 1 wieder herstellen

END:  LAR1  #AR1; // ursprüngliches Adressregister 1 herstellen


END_FUNCTION

FUNCTION "m7a_Collect_Nibble" : VOID
TITLE =Collect a Nibble (4 Bits)
//Collects 4 Bits as a Nibble
//
//----------------------------------------------------------------------
//Further Code to work wiht Nibbles
//
//How to Join 2 Nibbles as a single Byte
//
//L  bLowNibble    // load the Byte which should be the Low Nibble
//L  W#16#0F       // Set the 4 High Bits to 0
//UW
//L  bHighNibble   // load the Byte which should be the High Nibble
//SLW 4            // Shift it left 4 Bits
//OW
//T  TheByte
//----------------------------------------------------------------------
//
//AUTOR: Stefan Maag, Dipl.-Ing. (FH) Elektrotechnik
//DATUM: 7/2015
//INTERNET: www.maagic7.de
//
//AENDERUNGSVERMERKE:
//--------------------------------------------------------------------------------
//DATUM        NAME        AENDERUNG
//--------------------------------------------------------------------------------
//
//--------------------------------------------------------------------------------
//
//HINWEISE:
AUTHOR : 'S.Maag'
FAMILY : Maagic7
VERSION : 0.1


VAR_INPUT
  xIN1 : BOOL ;
  xIN2 : BOOL ;
  xIN3 : BOOL ;
  xIN4 : BOOL ;
END_VAR
VAR_OUTPUT
  xOut1 : BOOL ;	//= IN1
  xOut2 : BOOL ;	//= IN2
  xOut3 : BOOL ;	//= IN3
  xOut4 : BOOL ;	//= IN4
  bNibble : BYTE ;	//The Nibble: Bit 0..3
END_VAR
BEGIN
NETWORK
TITLE =

      L     0; // clear the first Temp-Byte
      T     LB     0;

      U     #xIN1; // collect the Bits
      =     #xOut1;
      =     L      0.0;

      U     #xIN2;
      =     #xOut2;
      =     L      0.1;

      U     #xIN3;
      =     #xOut3;
      =     L      0.2;

      U     #xIN4;
      =     #xOut4;
      =     L      0.3;

      L     LB     0; // write the Nibble
      T     #bNibble;

      SET   ;
      SAVE  ;
      CLR   ;


END_FUNCTION

FUNCTION "m7a_BitCount_uni" : INT
TITLE =BitCount: Zählt die Anzahl der Bits in Akku1 : BIE:= >0
//Zählt die Anzahl der Bits in AKKU1 und gibt diese als INT in RET_VAL zurück.
//Der zu prüfende Wert muss vorher in den AKKU1 geladen werden. Diese
//Vorgehensweise ermöglicht es, unabhängig vom DatenTyp die Bits zu prüfen, was
//mit einer Wertübergabe mittels eines Eingangsparamters des FC nicht möglich
//wäre.
//
//Die Anzahl der Bits stehen nach dem Bausteinaufruf auch im AKKU1 zur Verfügung
//und können von dort direkt weiterverarbeitet werden. Es ist also nicht zwingend
//notwendig, den Rückgabewert zu verwenden.
//
//(Hinweis: Durch den Bausteinaufruf wird der AKKU-Inhalt nicht verändert!)
//
//[CALL]
//immer Call verwenden, ein unbedingter aufruf mittels UC ist nicht möglich, da
//mit UC keine Paramterübergabe möglich ist und somit ein Fehler beim Schreiben
//des RET_VAL erfolgt.
//
//L  2#1100_0110         // 4 gesetzte Bits in AKKU1 laden
//CALL  "BitCount_uni"   // zählt die Bits
//       RET_VAL:=#Bits  // gibt die Anazhl (4) in Bits zurück
//
//L 2                    // da die Anzahl der Bits auch im AKKU1 enthalten sind
//>I                     // kann gleich direkt damit weitergearbeitet und z.B.
//="MoreThan2"           // auf mehr als 2 gesetzte Bits verglichen werden
//----------------------------------------------------------------------
//
//AUTOR: Stefan Maag, Dipl.-Ing. (FH) Elektrotechnik
//DATUM: 16/02/2003
//INTERNET: www.maagic7.de
//
//AENDERUNGSVERMERKE:
//--------------------------------------------------------------------------------
//DATUM       NAME       AENDERUNG
//--------------------------------------------------------------------------------
//31.07.2008  S.Maag     FC-ENO/BIE-Bit = High, wenn Anzahl der Bits >0
//                       Adressregister 1 sichern
//--------------------------------------------------------------------------------
//
//HINWEISE:
AUTHOR : 'S.Maag'
FAMILY : Maagic7
VERSION : 0.1


VAR_TEMP
  AR1 : DWORD ;
END_VAR
BEGIN
NETWORK
TITLE =Anzahl der gestzten Bits in Akku 1 Zählen
//Der Wert mit den zu zählenden Bits muss vorher in Akku 1 geladen werden.
//Die Anzahl der Bits wird dann in RET_VAL zurückgeben, steht aber auch noch
//zusätzlich im Akku1 zur Verfügung
      TAR1  #AR1; // Adressregister im TEMP-Bereich sichern
      L     0; // Adressregister 1 wird als BitZaehler verwendet
      LAR1  ; // daher auf 0 setzten
LOOP: TAK   ; // zu prüfende Bits wieder in Akku 1
      SRD   1; // erstes zu Prüfendes Bit hinausschieben
      SPZ   NEXT; // Wenn 0 dann Schleifenende prüfen
      +AR1  P#0.1; // Bitzähler im Adressregister 1 um 1 erhöhen
NEXT: L     0; // Vergleichswert, Bits zählen bis 0 erreicht
      <>D   ; // Solange wiederholen bis zu prüfende Bits
      SPB   LOOP; // den Wert 0 erreicht haben, alle Bits gezählt!
      TAR1  ; // Anzahl Bits aus Adressregister in Akku 1
      <>D   ; // Anzahl Bits auf 0 prüfen (mit vorheriger 0, bereits im AKKU)
      SAVE  ; // BIE-BIT = High, wenn Anzahl der Bits<>0
      CLR   ; // VKE wieder rücksetzen (verarbeiten)
      T     #RET_VAL; // Anzahl Bits in Rückgabewert
      LAR1  #AR1; // ursprüngliches Adressregister 1 wieder herstellen

END_FUNCTION

FUNCTION "m7a_BitCount_INT" : VOID
TITLE =zaehlt die gesetzten Bits in einem INT-Wert : BIE:= >0
//AUTOR: Stefan Maag, Dipl.-Ing. (FH) Elektrotechnik
//DATUM: 16/02/2003
//INTERNET: www.maagic7.de
//
//AENDERUNGSVERMERKE:
//--------------------------------------------------------------------------------
//DATUM       NAME       AENDERUNG
//--------------------------------------------------------------------------------
//31.07.2008  S.Maag     FC-ENO = High, wenn Bit gefunden, sonst LOW
//                       Adressregister 1 sichern
//--------------------------------------------------------------------------------
//
//HINWEISE:
AUTHOR : 'S.Maag'
FAMILY : Maagic7
VERSION : 0.1


VAR_INPUT
  Wert : INT ;	//zu prüfender Wert
END_VAR
VAR_OUTPUT
  Bits : INT ;	//anzahl gesetzter Bits
END_VAR
VAR_TEMP
  AR1 : DWORD ;
END_VAR
BEGIN
NETWORK
TITLE =Anzahl der gestzten Bits in INT Zählen
//Die Anzahl der Bits wird dann in #Bits zurückgeben, steht aber auch noch
//zusätzlich im Akku1 zur Verfügung
      TAR1  #AR1; // Adressregister im TMEP-Bereich sichern
      L     #Wert; // zu prüfenden Wert in Akku 1
      L     0; // Adressregister 1 wird als BitZaehler verwendet
      LAR1  ; // daher auf 0 setzten
LOOP: TAK   ; // zu prüfende Bits wieder in Akku 1
      SRD   1; // erstes zu Prüfendes Bit hinausschieben
      SPZ   NEXT; // Wenn 0 dann Schleifenende prüfen
      +AR1  P#0.1; // Bitzähler im Adressregister 1 um 1 erhöhen
NEXT: L     0; // Vergleichswert, Bits zählen bis 0 erreicht
      <>D   ; // Solange wiederholen bis zu prüfende Bits
      SPB   LOOP; // den Wert 0 erreicht haben, alle Bits gezählt!
      TAR1  ; // Anzahl Bits aus Adressregister in Akku 1
      <>D   ; // Anzahl Bits auf 0 prüfen (mit vorheriger 0, bereits im AKKU)
      SAVE  ; // BIE-BIT = High, wenn Anzahl der Bits<>0
      CLR   ; // VKE wieder rücksetzen (verarbeiten)
      T     #Bits; // Anzahl Bits in Rückgabewert
      LAR1  #AR1; // Adressregister wieder herstellen

NETWORK
TITLE =alternativer Code
//    // #BitCounter & #LoopRegister im TEMP-Bereich als INT anlegen
//
//      L     0
//      T     #BitCounter                 // Anzahl Bits auf 0
//      L     2#1000000000000000          // SchleifenRegister
//      T     #LoopRegister               // initialisieren
//
//      L     #Wert                       // zu prüfenden Wert in Akku 1
//loop: SRW   1                           // 1 Bit hinausschieben
//      SPP   inc                         // wenn positiv, dann Bit zaehlen
//      SPA   next                        // sonst weiter mit Schleifenregister
//
//inc:  L     #BitCounter                 // Bit zählen
//      +     1
//      T     #BitCounter
//      TAK                               // zu prüfenden Wert in Akku 1 zurück
//
//next: L     #LoopRegister               // SchleifenRegister auf nächstes Bit
//      SRW   1
//      SPP   end                         // falls positiv, dann letztes Bit !=
//Ende
//      T     #LoopRegister
//      TAK
//      SPA   loop
//
//end:  L     #BitCounter                 // Anzahl Bits zurückgeben
//      T     #Bits
//      L     0                           // BIE-Bit=High, wenn Anzahl Bits >0
//      <>I
//      SAVE
//      CLR
//


END_FUNCTION

FUNCTION "m7a_FirstBit_INT" : VOID
TITLE =sucht das erste gesetzte Bit in einem INT-Wert : BIE:= >0
//AUTOR: Stefan Maag, Dipl.-Ing. (FH) Elektrotechnik
//DATUM: 16/02/2003
//INTERNET: www.maagic7.de
//
//AENDERUNGSVERMERKE:
//--------------------------------------------------------------------------------
//DATUM       NAME       AENDERUNG
//--------------------------------------------------------------------------------
//31.07.2008  S.Maag     FC-ENO = High, wenn Bit gefunden, sonst LOW
//--------------------------------------------------------------------------------
//
//HINWEISE:
AUTHOR : 'S.Maag'
FAMILY : Maagic7
VERSION : 0.1


VAR_INPUT
  Value : INT ;	//zu prüfender Wert
END_VAR
VAR_OUTPUT
  BitPos : INT ;	//Position des ersten gesetzten Bits
END_VAR
BEGIN
NETWORK
TITLE =Nr des ersten gesetzten Bits

      L     #Value; // zu prüfenden Wert in Akku
      L     0; // vergleichen ob Wert = 0
      <>I   ; // dann Ende, wenn nicht muss mind. 1 Bit gesetzt sein
      SAVE  ; // Anzahl Bits <> 0 in BIE-Bit speichern
      SPBN  end; // ENDE, wenn Wert = 0
      INC   1; // Schleifenzaehler in Akku 1 auf 1 stellen = BitPosition
      TAK   ; // zu prüfende Bits in Akku 1 zurück
Loop: SRW   1; // 1 Bit hinausschieben
      SPP   save; // wenn poitiv, dann erstes Bit gefunden => speichern
      TAK   ; // Schleifenzaehler in Akku 1
      INC   1; // erhöhen Schleifenzaehler, BitNr.
      TAK   ; // zu prüfende Bits in Akku zurück
      SPA   Loop; // Schleife für nächstes Bit wiederholen
save: TAK   ; // Schleifenzaehler, BitNr in Akku 1
end:  T     #BitPos; // BitPosition zurückgeben


END_FUNCTION

FUNCTION "m7a_LastBit_INT" : VOID
TITLE =Nr.(1..16) letztes gesetzte Bit in einem INT-Wert (1..16)
//BIE := Bit gefunden, Position > 0
//
//[IN]
//Value  : Wert, von dem das letzte Bit ermittelt werden soll
//
//[OUT]
//BitPos : Position des letzten gesetzten Bits (1..16)
//         Es wird 0 zurückgegeben, wenn kein Bit gesetzt ist
//
//AUTOR: Stefan Maag, Dipl.-Ing. (FH) Elektrotechnik
//DATUM: 16/02/2003
//INTERNET: www.maagic7.de
//
//AENDERUNGSVERMERKE:
//--------------------------------------------------------------------------------
//DATUM       NAME       AENDERUNG
//--------------------------------------------------------------------------------
//31.07.2008  S.Maag     FC-ENO = High, wenn Bit gefunden, sonst LOW
//--------------------------------------------------------------------------------
//
//HINWEISE:
AUTHOR : 'S.Maag'
FAMILY : Maagic7
VERSION : 0.1


VAR_INPUT
  Value : INT ;	//zu prüfender Wert
END_VAR
VAR_OUTPUT
  BitPos : INT ;	//Position des ersten gesetzten Bits
END_VAR
BEGIN
NETWORK
TITLE =Nr des letzten gesetzten Bits

      L     #Value; // zu prüfenden Wert in Akku
      L     0; // vergleichen ob Wert = 0
      <>I   ; // dann Ende, wenn nicht muss mind. 1 Bit gesetzt sein
      SAVE  ; // Anzahl Bits <> 0 in BIE-Bit speichern
      SPBN  end; // ENDE, wenn Wert = 0
      INC   16; // Schleifenzaehler in Akku 1 auf 16 stellen = letzte BitPosition
      TAK   ; // zu prüfende Bits in Akku 1 zurück
Loop: SLW   1; // 1 Bit hinausschieben
      SPP   save; // wenn poitiv, dann letztes Bit gefunden => speichern
      TAK   ; // Schleifenzaehler in Akku 1
      DEC   1; // Schleifenzaehler erniedrigen, BitNr.
      TAK   ; // zu prüfende Bits in Akku zurück
      SPA   Loop; // Schleife für nächstes Bit wiederholen
save: TAK   ; // Schleifenzaehler, BitNr in Akku 1
end:  T     #BitPos; // BitPosition zurückgeben

END_FUNCTION

FUNCTION "m7a_BitGruppen_INT" : VOID
TITLE =zaehlt Bitgruppen in einem INT-Wert
//Autor:    Stefan Maag
//Datum:    12/1998 für S5
//          05/2002 für S7
//
//Zählt die Bitgruppen in einem Wert und gibt deren Anzahl zurück
//
//Bitgruppen werden begrenzt durch Wortanfang und Wortende sowie durch Nullen.
//Eine Bitgruppe besteht aus mindestens einer 1
//
//z.B.    1110 0001 0110 0010  enthält 4 Bitgruppen
//
//Funktion:  Druch negieren des Bitmusters werden Bitübergänge in genau negativer
//           weise zum Ausgangsmuster erzeugt. Verschiebt man diese beiden Muster
//           um 1 Bit gegeneinander, so entstehen genau an den Bitübergängen des
//           originals "1"-Paare. Diese Paare lassen sich durch den UW-Befehl
//           separieren. Zaehlt man nun die Bits nach dem Verunden, erhält man
//           die Anzahl der Bituebergänge im Ausgangswert. = Anzhal der Bitgruppen
//
//AUTOR: Stefan Maag, Dipl.-Ing. (FH) Elektrotechnik
//Datum:    12/1998 für S5
//          05/2002 für S7
//INTERNET: www.maagic7.de
//
//AENDERUNGSVERMERKE:
//--------------------------------------------------------------------------------
//DATUM      NAME        AENDERUNG
//--------------------------------------------------------------------------------
//
//--------------------------------------------------------------------------------
//
//HINWEISE:
AUTHOR : 'S.Maag'
FAMILY : Maagic7
VERSION : 0.1


VAR_INPUT
  Wert : INT ;	//auf Bitgruppen zu prüfender Wert
END_VAR
VAR_OUTPUT
  BitGruppen : INT ;	//Anzahl der enthaltenen Bitgruppen
END_VAR
VAR_TEMP
  BitCounter : INT ;
  LoopRegister : INT ;
END_VAR
BEGIN
NETWORK
TITLE =

      L     0;
      T     #BitCounter; // Anzahl Bits auf 0
      L     2#1000000000000000; // SchleifenRegister
      T     #LoopRegister; // initialisieren

      L     #Wert; // zu prüfenden Wert in Akku 1
      PUSH  ; // Wert auch in Akku 2 kopieren
      SRW   1; // fuer Übergänge Bits um 1 schieben
      INVI  ; // und negieren
      UW    ; // UW wertet die 0-1 Übergänge aus

// nun noch die Bits der 0-1 Übergänge zählen = Anzahl der Bitgruppen

loop: SRW   1; // 1 Bit hinausschieben
      SPP   inc; // wenn positiv, dann Bit zaehlen
      SPA   next; // sonst weiter mit Schleifenregister

inc:  L     #BitCounter; // Bit zählen
      +     1;
      T     #BitCounter;
      TAK   ; // zu prüfenden Wert in Akku 1 zurück

next: L     #LoopRegister; // SchleifenRegister auf nächstes Bit
      SRW   1;
      SPP   end; // falls positiv, dann letztes Bit != Ende
      T     #LoopRegister;
      TAK   ;
      SPA   loop;

end:  L     #BitCounter; // Anzahl Bits zurückgeben
      T     #BitGruppen;


NETWORK
TITLE =



END_FUNCTION

FUNCTION "m7b_ABS_DIFF_S7SysTime" : VOID
TITLE =ABS_DIFF_S7SysTime : Differenz zweier S7SystemZeiten 31Bit-Werte
//Da die S7 Systemzeit mittels SFC64 "TIME_TCK" nur 31 Bit 0..2147483647 ms
//aufweist gibt es einen Fehler, wenn Zeitdifferenzen über eine Timerüberlauf
//ermittelt werden. Um dies zu verhindern muss die Systemzeit auf 32Bit erweitert
//werden.
//
//Der Aufruf dieses FC ist für AWL vorgesehn, als Unconditioned Call
//
//L  #SysTime1
//L  #SysTime2
//UC FC 256
//T  #TimeDiff
//
//AUTOR: Stefan Maag, Dipl.-Ing. (FH) Elektrotechnik
//DATUM: 13/2013
//INTERNET: www.maagic7.de
//
//AENDERUNGSVERMERKE:
//--------------------------------------------------------------------------------
//DATUM        NAME       AENDERUNG
//--------------------------------------------------------------------------------
//15.01.2016   S.Maag     Fälschlich vorhandene IO-Paramter entfernt
//--------------------------------------------------------------------------------
//
//HINWEISE:
AUTHOR : 'S.Maag'
FAMILY : Maagic7
VERSION : 0.1


VAR_TEMP
  SysTimer : TIME ;
END_VAR
BEGIN
NETWORK
TITLE =die beiden Zeitwerte müssen bereits in den Akkus stehen

      SLD   1; // 1. Zeit in Akku 1 auf 32 Bit-Wert erweitern
      TAK   ; // Akkus tauschen
      SLD   1; // 2. Zeit auf 32 Bit-Wert erweitern
      -D    ; // Differenz bilden (=doppelte Differenz)
      SPPZ  pos; // If <0 THEN
      NEGD  ; //             'Vorzeichen umkehren'
pos:  SRD   1; // 32 Bit Korrektur wieder entferen TimeDiff nun in AKKU 1



END_FUNCTION

FUNCTION "TIME_SEC_TO_S5T" : VOID
TITLE =Zeiteingabe DINT mit varibalen Kommastellen -> S5Time
//Use this Function to replace the Siemens FC40 TIM_S5TI
AUTHOR : 'S.Maag'
VERSION : 0.1


VAR_INPUT
  diTime : DINT ;	//Zeiteingabe
  diFakt : DINT ;	//Faktor für Eingangszeit auf ms umrechnen (z.B. 100 bei Eingabe von x.x sec)
END_VAR
VAR_OUTPUT
  outS5T : S5TIME ;
END_VAR
VAR_TEMP
  bS5TimeBase : BYTE ;
  tmpTIME : DWORD ;
END_VAR
BEGIN
NETWORK
TITLE =
//S5-Timer is a  16Bit Value consisting of 3 BCD digits and a TimeBase
//
//   TimeBase.BCD3.BCD2.BCD1
//
//S5-Time Bases
//1/100sec  : 0
//1/10sec   : 1
//1 sec     : 2
//10sec     : 3
//
//FC-ENO: TRUE  : if no error
//        FALSE : Time is out of S5-Range: Timer output limited to the min/max
//                Value. S5T#0ms or S5T#9990s
      SET   ;
      SAVE  ;
      CLR   ;

      L     0; // Standard TimeBase 1/100sec
      T     #bS5TimeBase; // tmpByte := 0

      L     #diTime; // Time-Value Input
      L     #diFakt; // factor for Time Input
      *D    ;
      T     #tmpTIME; // Time  [ms]
      L     0;
      <D    ;
      SPB   ERR; // Error Time <0
      TAK   ;
      L     L#9990000; // max. Time S5-Timer  9990.000ms
      <=D   ;
      SPB   LOOP;
      L     W#16#3999; // Set Time to max. S5-Time 999*10sec
      SPB   ERR;
LOOP: L     #tmpTIME; // calculate Time-Value and TimeBase
      L     L#10;
      /D    ;
      T     #tmpTIME;
      L     L#999;
      <=D   ;
      SPB   END;
      L     #bS5TimeBase; // Next S5 Time Base [0/1/2/3]
      INC   1;
      T     #bS5TimeBase;
      SPA   LOOP; // LOOP UNTIL TimeBase is found
END:  TAK   ; // Get extracted TimeValue back to Akku1
      DTB   ; // convert 32Bit to BCD as S5Timer needs
      L     #bS5TimeBase; // the S5 TimeBase
      SLW   12; // shift the TimeBase to the left end of WORD
      OW    ; // join Time-Value and TimeBase to get S5-Timer-Format
      SPA   save; // READY
ERR:  CLR   ;
      SAVE  ;
save: T     #outS5T;
      BE    ;
END_FUNCTION

